// TIA Portal V19 export
FUNCTION "DEBUG_Test_Fun_Buffer_Topic1XX" : Void   // FC214, LAD
TITLE = TEST FUNZIONI BUFFER MESSAGGI
// stored: SetENOAutomatically false
   VAR_TEMP   // added for the SCL form of the ladder/FBD networks
      _w1 : Bool;
   END_VAR
BEGIN

REGION Network 1
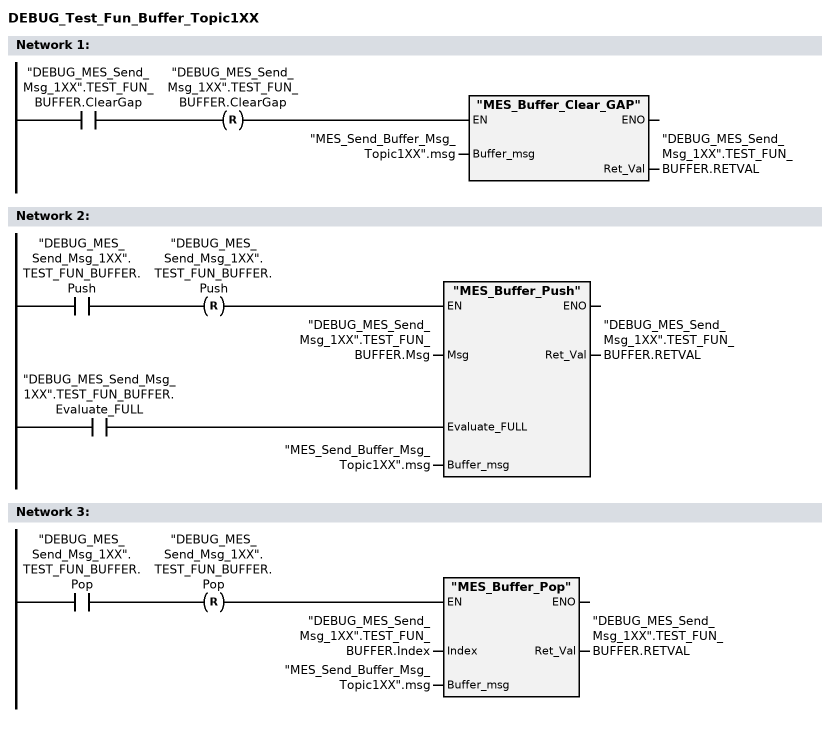
   RUNG wire#powerrail
      Contact( "DEBUG_MES_Send_Msg_1XX".TEST_FUN_BUFFER.ClearGap )
      R_Coil( "DEBUG_MES_Send_Msg_1XX".TEST_FUN_BUFFER.ClearGap )
      "MES_Buffer_Clear_GAP"(Buffer_msg := "MES_Send_Buffer_Msg_Topic1XX".msg, Ret_Val => "DEBUG_MES_Send_Msg_1XX".TEST_FUN_BUFFER.RETVAL)
   END_RUNG
   // the same network as SCL:
   #_w1 := "DEBUG_MES_Send_Msg_1XX".TEST_FUN_BUFFER.ClearGap;
   IF #_w1 THEN
       "DEBUG_MES_Send_Msg_1XX".TEST_FUN_BUFFER.ClearGap := FALSE;
       "DEBUG_MES_Send_Msg_1XX".TEST_FUN_BUFFER.RETVAL := "MES_Buffer_Clear_GAP"(Buffer_msg := "MES_Send_Buffer_Msg_Topic1XX".msg);
   END_IF;
END_REGION

REGION Network 2
   RUNG wire#powerrail
      Contact( "DEBUG_MES_Send_Msg_1XX".TEST_FUN_BUFFER.Push )
      R_Coil( "DEBUG_MES_Send_Msg_1XX".TEST_FUN_BUFFER.Push )
      "MES_Buffer_Push"(Evaluate_FULL := wire#w1, Msg := "DEBUG_MES_Send_Msg_1XX".TEST_FUN_BUFFER.Msg, Buffer_msg := "MES_Send_Buffer_Msg_Topic1XX".msg, Ret_Val => "DEBUG_MES_Send_Msg_1XX".TEST_FUN_BUFFER.RETVAL)
   END_RUNG
   RUNG wire#powerrail
      Contact( "DEBUG_MES_Send_Msg_1XX".TEST_FUN_BUFFER.Evaluate_FULL )
   END_RUNG wire#w1
   // the same network as SCL:
   #_w1 := "DEBUG_MES_Send_Msg_1XX".TEST_FUN_BUFFER.Push;
   IF #_w1 THEN
       "DEBUG_MES_Send_Msg_1XX".TEST_FUN_BUFFER.Push := FALSE;
       "DEBUG_MES_Send_Msg_1XX".TEST_FUN_BUFFER.RETVAL := "MES_Buffer_Push"(Msg := "DEBUG_MES_Send_Msg_1XX".TEST_FUN_BUFFER.Msg,
                               Evaluate_FULL := "DEBUG_MES_Send_Msg_1XX".TEST_FUN_BUFFER.Evaluate_FULL,
                               Buffer_msg := "MES_Send_Buffer_Msg_Topic1XX".msg);
   END_IF;
END_REGION

REGION Network 3
   RUNG wire#powerrail
      Contact( "DEBUG_MES_Send_Msg_1XX".TEST_FUN_BUFFER.Pop )
      R_Coil( "DEBUG_MES_Send_Msg_1XX".TEST_FUN_BUFFER.Pop )
      "MES_Buffer_Pop"(Index := "DEBUG_MES_Send_Msg_1XX".TEST_FUN_BUFFER.Index, Buffer_msg := "MES_Send_Buffer_Msg_Topic1XX".msg, Ret_Val => "DEBUG_MES_Send_Msg_1XX".TEST_FUN_BUFFER.RETVAL)
   END_RUNG
   // the same network as SCL:
   #_w1 := "DEBUG_MES_Send_Msg_1XX".TEST_FUN_BUFFER.Pop;
   IF #_w1 THEN
       "DEBUG_MES_Send_Msg_1XX".TEST_FUN_BUFFER.Pop := FALSE;
       "DEBUG_MES_Send_Msg_1XX".TEST_FUN_BUFFER.RETVAL := "MES_Buffer_Pop"(Index := "DEBUG_MES_Send_Msg_1XX".TEST_FUN_BUFFER.Index,
                               Buffer_msg := "MES_Send_Buffer_Msg_Topic1XX".msg);
   END_IF;
END_REGION
END_FUNCTION
